Staubli VAL3: refreshStatic.pgx

program refreshStatic()
  local num l_nSelected
  local num l_nSize
  local string l_sEvent
  local num l_nLocal
  local num i
  local string l_sMessage
begin
  cls()
  //
  // set the view of the page..
  //
  // set small x_nView
  call use:setView(false)
  // SET THE PAGE NUMBER
  use:nPage=100
  // USE <>PROFILE for <>PAGE
  use:nPage=use:nPage+abs(limit(saveData:mode,0,2)-2)
  //
  if cycleStatus:bCycle
    use:nPage=use:nPage+3
  endIf
  // load the menu page
  if saveData:language!="japanese"
    // SET THE VIEW OF THE PAGE
    call language:page(l_sMessage,use:nPage)
    // define the menu
    call use:stringToArray(l_sMessage,sMenu)
  else
    // japanese use the array for the menu
    call language:page(sMenu8,use:nPage)
    call use:stringCopy(sMenu8,sMenu)
  endIf
  if saveData:language!="japanese"
    call use:setMenu(sMenu,true,3)
  else
    call use:setMenu(sMenu,false,3)
  endIf
  call use:getMenu(sMenu,bButton)
  // use ON / OFF for the active gun
  bButton[2]=true
  call use:typeMenu(3,"")
  //
  call use:setSizeList(19,0,19,11)
  //
  // BUILD THE LIST
  //
  switch nProgID
    case 0
      call language:message(l_sMessage,25)
    break
    case 1
      l_sMessage="SUB-PROG"
    break
    case 2
      call language:message(l_sMessage,26)
    break
  endSwitch
  call use:listcreate(l_sMessage)
  call use:listadd(sList)
  call use:selectNewField(nSelected,nIndex,nView)
  nSelected=-1
  // is a filter using ??
  call language:message(l_sMessage,64)
  if saveData:sProgFilter!=""
    call use:type(0,1,l_sMessage+">"+saveData:sProgFilter)
  else
    call use:typeLen(0,1,"",len(l_sMessage+">"+saveData:sProgFilter))
  endIf
end
